PROGRAM MAIN
VAR
END_VAR

END_PROGRAM

(* stored: Version 1.1.0.1
   POU MAIN: Id {c1f1d386-8cc3-46ed-9ed3-aea6bd0dd0b2} *)
